// TIA Portal V17 export
// export: Created 2024-08-09T12:53:19.2323593Z, ExportSetting WithDefaults, DisplayName Totally Integrated Automation Portal, DisplayVersion V17 Update 7, DisplayName TIA Portal Openness, DisplayVersion V17 Update 7, DisplayName TIA Portal Version Control Interface, DisplayVersion V17, DisplayName STEP 7 Professional, DisplayVersion V17 Update 7, DisplayName STEP 7 Safety, DisplayVersion V17 Update 6, DisplayName WinCC Professional, DisplayVersion V17 Update 7
TYPE "S_Lanc_Exp"
// stored: IsFailsafeCompliant false
   STRUCT
      Pt_Zs : "S_Suivi_Dosage";
      CommunDos : "S_Dosage_Commun";
      Pt_Cel : "S_Cellule";
      Exp1 : "S_Exp_Dos";
      Exp2 : "S_Exp_Dos";
      Fg_Dest_Interm : Bool;
      Num_Ligne : SInt;
      Tac_Exp_Dos1 : SInt := -1;
      Tac_Exp_Dos2 : SInt := -1;
      Fg_Ctrl_Hop : Bool;
      Fg_Ctrl_Stock : Bool;
      Fg_Ctrl_Incomp : Bool;
      Fg_Ctrl_Incorp : Bool;
      Fg_Ench_Exp : Bool;
      Fg_Valid_Ench_NB : Bool;
      Fg_Valid_Deux_Cir : Bool;
      Fg_Chg_Dest_Serie_Dem_Cir : Bool;
      Memo_Circuit : SInt;
      Dial_Def : "S_DIALOG_DEF";
      Lst_Taches_Att_Chg_Exp : Array[0.."T_MAX_AMONTAVAL"] of "S_TacheNiv";
      Lst_Taches_Att_Fin_Prd_Sous_Mel : Array[0.."T_MAX_AMONTAVAL"] of "S_TacheNiv";
      Lst_Taches_Att_Fin_NB_Sous_Mel : Array[0.."T_MAX_AMONTAVAL"] of "S_TacheNiv";
      Lst_Taches_Aut_Ench : Array[0.."T_MAX_AMONTAVAL"] of "S_TacheNiv";
   END_STRUCT;
END_TYPE
